// Mitsubishi GX Works2 project: b10   PLC: Q02/Q02H

PROGRAM MAIN
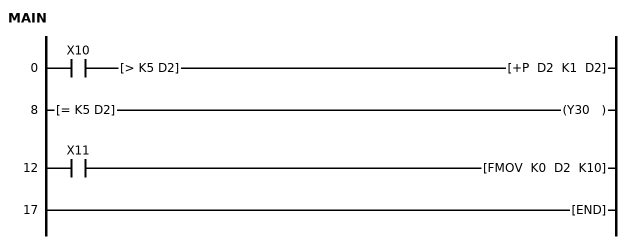
0     LD      X10
      AND>    K5 D2
      +P      D2 K1 D2
8     LD=     K5 D2
      OUT     Y30
12    LD      X11
      FMOV    K0 D2 K10
17    END
END_PROGRAM
